// Block: MwFakCalc_PERS

DATA_BLOCK MwFakCalc_PERS
VERSION : 0.1
   NON_RETAIN
   VAR
      PersistentValues : udt_MwFacCalc_Pers;
   END_VAR

BEGIN
   // No initialization required
END_DATA_BLOCK
